{attribute 'GeneratedUsingTerminal: EL3204-0200-0016'}
{attribute addProperty BoxType "EL3204-0200-0016"}
{attribute addProperty Id "StatusAT %I*Status_68C33E995ValueAT %I*INT2"}
{attribute addProperty CRC "2507538081"}
{attribute addProperty Size "7"}
TYPE RTD_Inputs_Channel_9575FEA1 :
STRUCT
	{attribute addProperty Name "Status"}
	Status AT %I* : Status_68C33E99;
	{attribute addProperty Name "Value"}
	Value AT %I* : INT;
END_STRUCT
END_TYPE

(* stored: Version 1.2.0.0, ProductVersion 3.1.4024.9
   DUT RTD_Inputs_Channel_9575FEA1: Id {a22ff471-1c4f-45f2-bd62-a5fc76d14def} *)
